// TIA Portal project "Convey1_4S" (V13)

(* hardware
DEVICE "S7300/ET200M-Station_1"  S7-300 station
   slot 0: "Profilschiene_0"  Rail  6ES7 390-1***0-0AA0
   slot 1: "PS 307 5A_1"  PS 307 5A  6ES7 307-1EA00-0AA0
   slot 2: "SIMATIC S7-300"  CPU 314C-2 PN/DP  6ES7 314-6EH04-0AB0  V3.3
      slot 2: "PROFINET-Schnittstelle_1"  PN-IO
         slot 1: "Port_1"  Port
         slot 2: "Port_2"  Port
      slot 5: "DI 24/DO 16_1"  DI24/DO16
      slot 6: "AI 5/AO 2_1"  AI5/AO2
      slot 7: "Zählen_1"  Counter
      slot 8: "Positionieren_1"  Positioning
   slot 4: "CP 343-2_1"  CP 343-2  6GK7 343-2AH01-0XA0  V3.1
*)

// ===== PLC "SIMATIC S7-300"  CPU 314C-2 PN/DP =====

VAR_GLOBAL   // PLC tag table "Standard-Variablentabelle"
   "Mx_Clock10Hz" AT %M100.0 : Bool;   // CPU clock memory-flag 0: f = 10 Hz / T = 0,1 s
   "Mx_Clock5Hz" AT %M100.1 : Bool;   // CPU clock memory-flag 1: f = 5 Hz / T = 0,2 s
   "Mx_Clock2,5Hz" AT %M100.2 : Bool;   // CPU clock memory-flag 2: f = 2,5 Hz / T = 0,4 s
   "Mx_Clock2Hz" AT %M100.3 : Bool;   // CPU clock memory-flag 3: f = 2 Hz / T = 0,5 s
   "Mx_Clock1,25Hz" AT %M100.4 : Bool;   // CPU clock memory-flag 4: f = 1,25 Hz / T = 0,8 s
   "Mx_Clock1Hz" AT %M100.5 : Bool;   // CPU clock memory-flag 5: f = 1 Hz / T = 1 s
   "Mx_Clock0,625Hz" AT %M100.6 : Bool;   // CPU clock memory-flag 6: f = 0,625 Hz / T = 1,6 s
   "Mx_Clock0,5Hz" AT %M100.7 : Bool;   // CPU clock memory-flag 7: f = 0,5 Hz / T = 2 s
   "Ix_S0_OFF" AT %I124.0 : Bool;   // OFF (NC)
   "Ix_S1_StartConveyor1" AT %I124.1 : Bool;   // Start conveyor 1
   "Ix_S2_StartConveyor2" AT %I124.2 : Bool;   // Start conveyor 2
   "Mx_Step1" AT %M10.0 : Bool;   // Grafcet, step-flag 1
   "Mx_Step2" AT %M10.1 : Bool;   // Grafcet, step-flag 2
   "Mx_Step10" AT %M10.2 : Bool;   // Grafcet, step-flag 10
   "Mx_Step11" AT %M10.3 : Bool;   // Grafcet, step-flag 11
   "Mx_Step12" AT %M10.4 : Bool;   // Grafcet, step-flag 12
   "Mx_Step13" AT %M10.5 : Bool;   // Grafcet, step-flag 13
   "Mx_Step14" AT %M10.6 : Bool;   // Grafcet, step-flag 14
   "Mx_StartingFlag" AT %M20.0 : Bool;   // Starting flag to activate the sequence (step 1)
   "Mx_PEdgeFlag_Step1" AT %M20.1 : Bool;   // Positive edge flag is activated when step 1 is activated
   "Mb_FlagByte10" AT %MB10 : Byte;   // Flag byte 10
   "Ix_S3_StartConveyor3" AT %I124.3 : Bool;   // Start conveyor 3
   "Qx_Q1_Conveyor1_ON" AT %Q124.0 : Bool;   // Conveyor 1 ON
   "Ix_S4_Enable" AT %I124.4 : Bool;   // Enable signal
   "Ix_F4-F5-F6(S5)" AT %I124.5 : Bool;   // Overload relay (NC)
   "Mx_PEdgeFlag_S4" AT %M20.2 : Bool;   // Positive edge flag is activated on pressing S4
   "Qx_Q2_Conveyor2_ON" AT %Q124.1 : Bool;   // Conveyor 2 ON
   "Qx_Q3_Conveyor3_ON" AT %Q124.2 : Bool;   // Conveyor 3 ON
   "Qx_P4_EnableActivated" AT %Q124.3 : Bool;   // Signal lamp "enable activated"
END_VAR

FUNCTION "Grafcet G1" : Void   // FC1, FBD
TITLE = Function diagram G1 (Grafcet)
{ S7_Optimized_Access := 'FALSE' }
VERSION : 0.1
// Programming of the function diagram (Grafcet)
   VAR_TEMP   // added for the SCL form of the ladder/FBD networks
      _w1 : Bool;
   END_VAR
BEGIN

REGION Network 1: Step 1
   // A dominant setting self-latching relay must be used. The step 1 cannot be set if step 2 is already active.
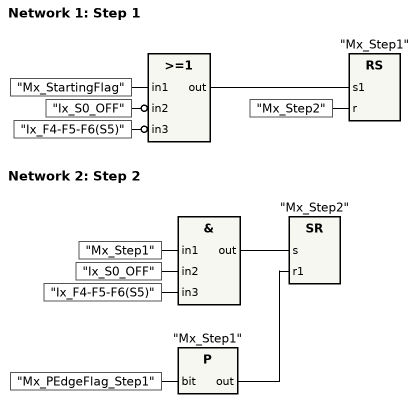
   IF "Mx_Step2" THEN
       "Mx_Step1" := FALSE;   // RS flip-flop
   END_IF;
   IF "Mx_StartingFlag" OR NOT "Ix_S0_OFF" OR NOT "Ix_F4-F5-F6(S5)" THEN "Mx_Step1" := TRUE; END_IF;
END_REGION

REGION Network 2: Step 2
   #_w1 := "Mx_Step1" AND NOT "Mx_PEdgeFlag_Step1";   // rising edge of "Mx_Step1"
   "Mx_PEdgeFlag_Step1" := "Mx_Step1";
   IF "Mx_Step1" AND "Ix_S0_OFF" AND "Ix_F4-F5-F6(S5)" THEN
       "Mx_Step2" := TRUE;   // SR flip-flop
   END_IF;
   IF #_w1 THEN "Mx_Step2" := FALSE; END_IF;
END_REGION
END_FUNCTION

FUNCTION "Grafcet G10" : Void   // FC2, FBD
TITLE = Function diagram G10 (Grafcet)
{ S7_Optimized_Access := 'FALSE' }
VERSION : 0.1
// Programming of the function diagram (Grafcet)
BEGIN

REGION Network 1: Step 10
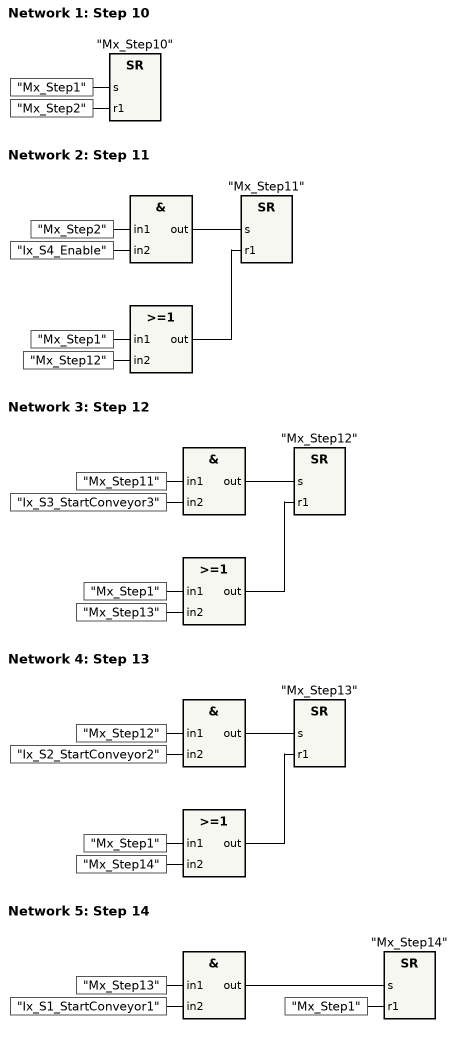
   IF "Mx_Step1" THEN
       "Mx_Step10" := TRUE;   // SR flip-flop
   END_IF;
   IF "Mx_Step2" THEN "Mx_Step10" := FALSE; END_IF;
END_REGION

REGION Network 2: Step 11
   IF "Mx_Step2" AND "Ix_S4_Enable" THEN
       "Mx_Step11" := TRUE;   // SR flip-flop
   END_IF;
   IF "Mx_Step1" OR "Mx_Step12" THEN "Mx_Step11" := FALSE; END_IF;
END_REGION

REGION Network 3: Step 12
   IF "Mx_Step11" AND "Ix_S3_StartConveyor3" THEN
       "Mx_Step12" := TRUE;   // SR flip-flop
   END_IF;
   IF "Mx_Step1" OR "Mx_Step13" THEN "Mx_Step12" := FALSE; END_IF;
END_REGION

REGION Network 4: Step 13
   IF "Mx_Step12" AND "Ix_S2_StartConveyor2" THEN
       "Mx_Step13" := TRUE;   // SR flip-flop
   END_IF;
   IF "Mx_Step1" OR "Mx_Step14" THEN "Mx_Step13" := FALSE; END_IF;
END_REGION

REGION Network 5: Step 14
   IF "Mx_Step13" AND "Ix_S1_StartConveyor1" THEN
       "Mx_Step14" := TRUE;   // SR flip-flop
   END_IF;
   IF "Mx_Step1" THEN "Mx_Step14" := FALSE; END_IF;
END_REGION
END_FUNCTION

FUNCTION "Actions" : Void   // FC3, FBD
TITLE = Execute the actions
{ S7_Optimized_Access := 'FALSE' }
VERSION : 0.1
BEGIN

REGION Network 1: Control conveyor 1 and signal lamp P1
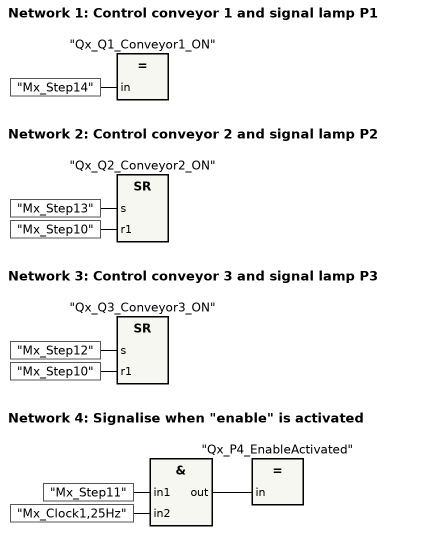
   "Qx_Q1_Conveyor1_ON" := "Mx_Step14";
END_REGION

REGION Network 2: Control conveyor 2 and signal lamp P2
   IF "Mx_Step13" THEN
       "Qx_Q2_Conveyor2_ON" := TRUE;   // SR flip-flop
   END_IF;
   IF "Mx_Step10" THEN "Qx_Q2_Conveyor2_ON" := FALSE; END_IF;
END_REGION

REGION Network 3: Control conveyor 3 and signal lamp P3
   IF "Mx_Step12" THEN
       "Qx_Q3_Conveyor3_ON" := TRUE;   // SR flip-flop
   END_IF;
   IF "Mx_Step10" THEN "Qx_Q3_Conveyor3_ON" := FALSE; END_IF;
END_REGION

REGION Network 4: Signalise when "enable" is activated
   "Qx_P4_EnableActivated" := "Mx_Step11" AND "Mx_Clock1,25Hz";
END_REGION
END_FUNCTION

ORGANIZATION_BLOCK "Main"   // OB1, FBD
TITLE = "Main Program Sweep (Cycle)"
{ S7_Optimized_Access := 'FALSE' }
VERSION : 0.1
// Organisation block OB1 is executed cyclically
BEGIN

REGION Network 1: Call the function diagram block G1
   // Programming of the function diagram (Grafcet)
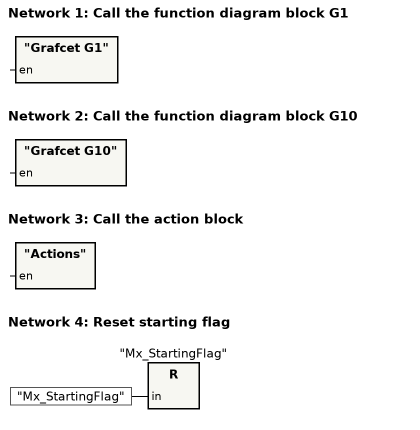
   "Grafcet G1"();
END_REGION

REGION Network 2: Call the function diagram block G10
   // Programming of the function diagram (Grafcet)
   "Grafcet G10"();
END_REGION

REGION Network 3: Call the action block
   // Programming of the actions
   "Actions"();
END_REGION

REGION Network 4: Reset starting flag
   IF "Mx_StartingFlag" THEN "Mx_StartingFlag" := FALSE; END_IF;
END_REGION
END_ORGANIZATION_BLOCK

ORGANIZATION_BLOCK "COMPLETE RESTART"   // OB100, FBD
TITLE = "Complete Restart"
{ S7_Optimized_Access := 'FALSE' }
VERSION : 0.1
// OB 100 is executed once only when the status of the PLC changes from STOP to RUN.
BEGIN

REGION Network 1: Reset flag byte 10 (step-flags)
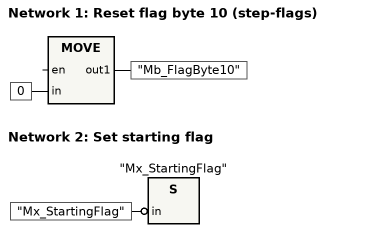
   "Mb_FlagByte10" := 0;
END_REGION

REGION Network 2: Set starting flag
   IF NOT "Mx_StartingFlag" THEN "Mx_StartingFlag" := TRUE; END_IF;
END_REGION
END_ORGANIZATION_BLOCK